// TIA Portal project "Motor-Direction-Control" (V18)

(* hardware
DEVICE "S7-1200 station_1"  S7-1200 Station
   slot 0: "Rack_0"  S7-1200 Rack  Rack  V1.0
   slot 1: "PLC_1"  CPU 1212C DC/DC/Rly  6ES7 212-1HE40-0XB0  V4.6
*)

// ===== PLC "PLC_1"  CPU 1212C DC/DC/Rly =====

VAR_GLOBAL   // PLC tag table "Default tag table"
   "startR" AT %I0.0 : Bool;
   "startL" AT %I0.1 : Bool;
   "stop" AT %I0.2 : Bool;
   "motorR" AT %Q0.0 : Bool;
   "motorL" AT %Q0.1 : Bool;
   "Tag_1" AT %M0.0 : Bool;
   "Tag_2" AT %M0.1 : Bool;
   "Tag_3" AT %M0.2 : Bool;
   "Tag_4" AT %M0.3 : Bool;
END_VAR

// folder: System blocks/Program resources

DATA_BLOCK "IEC_Timer_0_DB"   // DB1
{ S7_Optimized_Access := 'TRUE' }
AUTHOR : Simatic
FAMILY : IEC
NAME : IEC_TMR
VERSION : 1.0
// stored: InstanceOfName IEC_TIMER
"IEC_TIMER"
BEGIN
END_DATA_BLOCK

// folder: (top level)

ORGANIZATION_BLOCK "Main"   // OB1, LAD, ProgramCycle
TITLE = "Main Program Sweep (Cycle)"
{ S7_Optimized_Access := 'TRUE' }
VERSION : 0.1
   VAR_INPUT
      Initial_Call : Bool;   // Initial call of this OB
      Remanence : Bool;   // =True, if remanent data are available
   END_VAR
   VAR_TEMP   // added for the SCL form of the ladder/FBD networks
      _w1 : Bool;
      _w2 : Bool;
   END_VAR
BEGIN

REGION Network 1
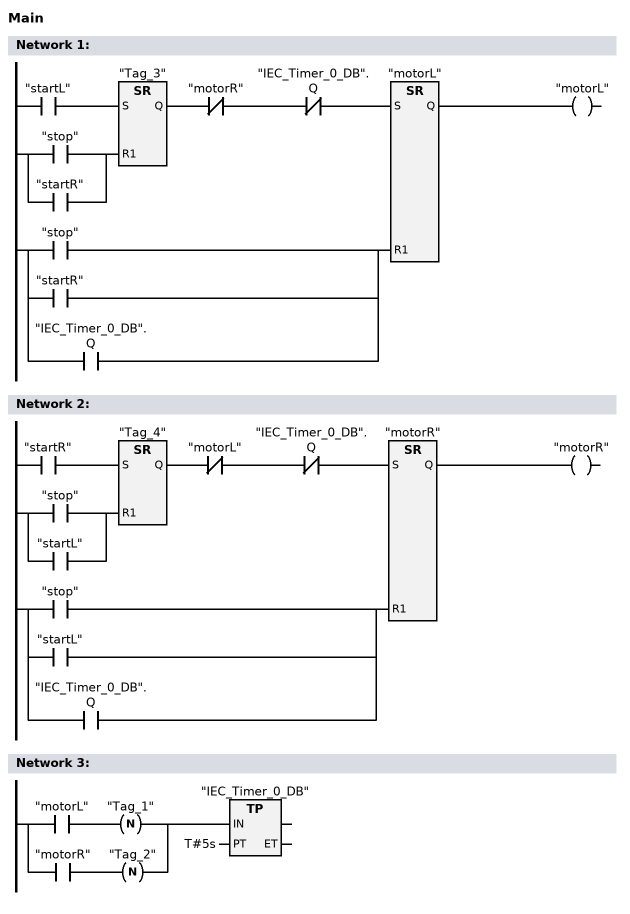
   RUNG wire#powerrail
      Contact( "startL" )
      S_SR(operand := "Tag_3", r1 := wire#w1)
      I_Contact( "motorR" )
      I_Contact( "IEC_Timer_0_DB".Q )
      S_SR(operand := "motorL", r1 := wire#w2)
      Coil( "motorL" )
   END_RUNG
   RUNG wire#powerrail
      Contact( "stop" )
   END_RUNG wire#w1
   RUNG wire#powerrail
      Contact( "startR" )
   END_RUNG wire#w1
   RUNG wire#powerrail
      Contact( "stop" )
   END_RUNG wire#w2
   RUNG wire#powerrail
      Contact( "startR" )
   END_RUNG wire#w2
   RUNG wire#powerrail
      Contact( "IEC_Timer_0_DB".Q )
   END_RUNG wire#w2
   // the same network as SCL:
   IF "startL" THEN
       "Tag_3" := TRUE;   // SR flip-flop
   END_IF;
   IF "stop" OR "startR" THEN "Tag_3" := FALSE; END_IF;
   IF "Tag_3" AND NOT "motorR" AND NOT "IEC_Timer_0_DB".Q THEN
       "motorL" := TRUE;   // SR flip-flop
   END_IF;
   IF "stop" OR "startR" OR "IEC_Timer_0_DB".Q THEN "motorL" := FALSE; END_IF;
   "motorL" := "motorL";
END_REGION

REGION Network 2
   RUNG wire#powerrail
      Contact( "startR" )
      S_SR(operand := "Tag_4", r1 := wire#w1)
      I_Contact( "motorL" )
      I_Contact( "IEC_Timer_0_DB".Q )
      S_SR(operand := "motorR", r1 := wire#w2)
      Coil( "motorR" )
   END_RUNG
   RUNG wire#powerrail
      Contact( "stop" )
   END_RUNG wire#w1
   RUNG wire#powerrail
      Contact( "startL" )
   END_RUNG wire#w1
   RUNG wire#powerrail
      Contact( "stop" )
   END_RUNG wire#w2
   RUNG wire#powerrail
      Contact( "startL" )
   END_RUNG wire#w2
   RUNG wire#powerrail
      Contact( "IEC_Timer_0_DB".Q )
   END_RUNG wire#w2
   // the same network as SCL:
   IF "startR" THEN
       "Tag_4" := TRUE;   // SR flip-flop
   END_IF;
   IF "stop" OR "startL" THEN "Tag_4" := FALSE; END_IF;
   IF "Tag_4" AND NOT "motorL" AND NOT "IEC_Timer_0_DB".Q THEN
       "motorR" := TRUE;   // SR flip-flop
   END_IF;
   IF "stop" OR "startL" OR "IEC_Timer_0_DB".Q THEN "motorR" := FALSE; END_IF;
   "motorR" := "motorR";
END_REGION

REGION Network 3
   #_w1 := NOT "motorL" AND "Tag_1";   // falling edge
   "Tag_1" := "motorL";
   #_w2 := NOT "motorR" AND "Tag_2";   // falling edge
   "Tag_2" := "motorR";
   "IEC_Timer_0_DB".TP(IN := #_w1 OR #_w2, PT := T#5s);
END_REGION
END_ORGANIZATION_BLOCK